(* IEC 61131-3 sources: dynamics/src/Dynamics, 9 files *)

(* ---- IDynamic.st ---- *)
NAMESPACE Simatic.Ax.Dynamics

    /// `Next(value)`
    INTERFACE IDynamic

        /// Pass process value
        /// Get next output
        METHOD Next : LREAL
            VAR_INPUT
                value : LREAL;
            END_VAR
        END_METHOD

    END_INTERFACE
END_NAMESPACE

(* ---- IOutputDynamic.st ---- *)
NAMESPACE Simatic.Ax.Dynamics
    /// `SetOutput`, extends `IDynamic, IOutputProvider`
    INTERFACE IOutputDynamic EXTENDS IDynamic, IOutputProvider
        /// Set output value
        /// New value should be used as base for next output
        METHOD SetOutput : LREAL
            VAR_INPUT
                output : LREAL;
            END_VAR
        END_METHOD
    END_INTERFACE
END_NAMESPACE

(* ---- Amplifier.st ---- *)
NAMESPACE Simatic.Ax.Dynamics
    CLASS Amplifier IMPLEMENTS IDynamic

        /// Amplification
        VAR PUBLIC
            k : LREAL := 1.0;
        END_VAR

        /// Get amplification
        METHOD PUBLIC GetK : LREAL
            GetK := k;
        END_METHOD
        /// Set ampflification
        METHOD PUBLIC SetK
            VAR_INPUT
                newK : LREAL;
            END_VAR
            k := newK;
        END_METHOD

        METHOD PUBLIC Next : LREAL
            VAR_INPUT
                value : LREAL;
            END_VAR
            Next := k * value;
        END_METHOD

    END_CLASS
END_NAMESPACE

(* ---- BoundedOutputDynamic.st ---- *)
NAMESPACE Simatic.Ax.Dynamics
    CLASS BoundedOutputDynamic EXTENDS BoundedDynamic IMPLEMENTS IOutputDynamic

        VAR PRIVATE
            _storingDynamic : IOutputDynamic;
        END_VAR

        METHOD PUBLIC SetUnboundedDynamic
            VAR_INPUT
                newDynamic : IOutputDynamic;
            END_VAR
            _storingDynamic := newDynamic;
            unboundedDynamic := _storingDynamic;
        END_METHOD

        METHOD PUBLIC GetOutput : LREAL
            GetOutput := _storingDynamic.GetOutput();
        END_METHOD
        METHOD PUBLIC SetOutput : LREAL
            VAR_INPUT
                output : LREAL;
            END_VAR
            SetOutput := _storingDynamic.SetOutput(output);
        END_METHOD

        METHOD PUBLIC OVERRIDE Next : LREAL
            VAR_INPUT
                value : LREAL;
            END_VAR
            Next := _storingDynamic.SetOutput(SUPER.Next(value));
        END_METHOD

        METHOD PUBLIC IsMin : BOOL
            IsMin := _storingDynamic.GetOutput() = THIS.GetMinOutput();
        END_METHOD
        METHOD PUBLIC IsMax : BOOL
            IsMax := _storingDynamic.GetOutput() = THIS.GetMaxOutput();
        END_METHOD

    END_CLASS
END_NAMESPACE

(* ---- Differentiator.st ---- *)
NAMESPACE Simatic.Ax.Dynamics
    CLASS Differentiator EXTENDS FirstOrderDynamic

        VAR PUBLIC
            /// Lead time in seconds
            tDSeconds : LREAL;
        END_VAR

        VAR PRIVATE
            _value : LREAL;
        END_VAR

        /// Get lead time in seconds
        METHOD PUBLIC GetTDSeconds : LREAL
            GetTDSeconds := tDSeconds;
        END_METHOD
        /// Set lead time in seconds
        METHOD PUBLIC SetTDSeconds
            VAR_INPUT
                newTDSeconds : LREAL;
            END_VAR
            tDSeconds := newTDSeconds;
        END_METHOD
        /// Set lead time in seconds and amplification
        /// SetTDSeconds(newTDSeconds, k) is equivalent to SetTDSeconds(newTDSeconds * k)
        METHOD PUBLIC SetTDSeconds
            VAR_INPUT
                newTDSeconds : LREAL;
                k : LREAL;
            END_VAR
            THIS.SetTDSeconds(newTDSeconds * k);
        END_METHOD

        /// Get last process value
        METHOD INTERNAL GetValue : LREAL
            GetValue := _value;
        END_METHOD

        METHOD PROTECTED OVERRIDE _Next : LREAL
            VAR_INPUT
                value : LREAL;
                elapsedSeconds : LREAL;
            END_VAR
            _Next := (value - _value) / elapsedSeconds * tDSeconds;
            _value := value;
        END_METHOD

    END_CLASS
END_NAMESPACE

(* ---- FirstOrderDynamic.st ---- *)
NAMESPACE Simatic.Ax.Dynamics
    /// Dynamic exploiting the elapsed time since last call
    /// `elapsedTimeProvider` must be given!
    CLASS INTERNAL ABSTRACT FirstOrderDynamic IMPLEMENTS IDynamic

        VAR PUBLIC
            /// Provides elapsed time since last call to `Next()`
            /// `elapsedTimeProvider.Start()` will be called automatically on `Next()`
            /// User should never call `elapsedTimeProvider.Start()`!
            /// Unexpected behaviour could be the result.
            elapsedTimeProvider : IElapsedSecondsProvider;
        END_VAR

        /// Maps the process value and the elapsed time in seconds to the next output value
        METHOD PROTECTED ABSTRACT _Next : LREAL
            VAR_INPUT
                value : LREAL;
                elapsedSeconds : LREAL;
            END_VAR
        END_METHOD
        METHOD PUBLIC FINAL Next : LREAL
            VAR_INPUT
                value : LREAL;
            END_VAR
            Next := this._Next(value, elapsedTimeProvider.GetElapsedSeconds());
            elapsedTimeProvider.Start();
        END_METHOD

    END_CLASS
END_NAMESPACE

(* ---- FirstOrderOutputDynamic.st ---- *)
NAMESPACE Simatic.Ax.Dynamics
    /// Dynamic exploiting the elapsed time since last call and last output value
    /// `elapsedTimeProvider` must be given!
    CLASS INTERNAL ABSTRACT FirstOrderOutputDynamic EXTENDS FirstOrderDynamic IMPLEMENTS IOutputDynamic

        VAR PRIVATE
            _output : LREAL;
        END_VAR

        METHOD PUBLIC GetOutput : LREAL
            GetOutput := _output;
        END_METHOD
        METHOD PUBLIC SetOutput : LREAL
            VAR_INPUT
                output : LREAL;
            END_VAR
            _output := output;
            SetOutput := _output;
        END_METHOD

        /// Maps process value, elapsed time since last call and last output value to next output value
        METHOD PROTECTED ABSTRACT _Next : LREAL
            VAR_INPUT
                value : LREAL;
                elapsedSeconds : LREAL;
                output : LREAL;
            END_VAR
        END_METHOD

        METHOD PROTECTED FINAL OVERRIDE _Next : LREAL
            VAR_INPUT
                value : LREAL;
                elapsedSeconds : LREAL;
            END_VAR
            _Next := this.SetOutput(this._Next(value, elapsedSeconds, _output));
        END_METHOD

    END_CLASS
END_NAMESPACE

(* ---- IdentityDynamic.st ---- *)
NAMESPACE Simatic.Ax.Dynamics
    CLASS IdentityDynamic IMPLEMENTS IDynamic

        METHOD PUBLIC Next : LREAL
            VAR_INPUT
                value : LREAL;
            END_VAR
            Next := value;
        END_METHOD

    END_CLASS
END_NAMESPACE

(* ---- ParallelFirstOrderDynamic.st ---- *)
NAMESPACE Simatic.Ax.Dynamics
    /// The process value is passed to two first order dynamics.
    /// The output values are summed up and multiplied by the factor K.
    CLASS INTERNAL ABSTRACT ParallelFirstOrderDynamic EXTENDS FirstOrderDynamic

        VAR PUBLIC
            /// The factor K
            k : LREAL := 1.0;
        END_VAR

        VAR PROTECTED
            /// Provides the time of the real time provider in the moment of the call to next.
            /// The use of a pseudo time provider ensures the same elapsed time is used by both dynamics.
            /// Moreover, time is saved by not calling the measuring function twice.
            _pseudoTimeProvider : ConstantTimeProvider;
        END_VAR

        /// Get the factor K
        METHOD PUBLIC GetK : LREAL
            GetK := k;
        END_METHOD
        /// Set the factor K
        METHOD PUBLIC SetK
            VAR_INPUT
                newK : LREAL;
            END_VAR
            k := newK;
        END_METHOD

        /// The method `Next` of one dynamic
        METHOD PROTECTED ABSTRACT _Next0 : LREAL
            VAR_INPUT
                value : LREAL;
            END_VAR
        END_METHOD
        /// The method `Next` of the other dynamic
        METHOD PROTECTED ABSTRACT _Next1 : LREAL
            VAR_INPUT
                value : LREAL;
            END_VAR
        END_METHOD

        METHOD PROTECTED FINAL OVERRIDE _Next : LREAL
            VAR_INPUT
                value : LREAL;
                elapsedSeconds : LREAL;
            END_VAR
            _pseudoTimeProvider.seconds := elapsedSeconds;
            _Next := k * (this._Next0(value) + this._Next1(value));
        END_METHOD

    END_CLASS
END_NAMESPACE
